PROGRAM AxisReset
VAR
END_VAR

//左臂
axis_LeftArm_Left_Reset(
	Axis:= axis_LeftArm_Left, 
	Execute:= bAxis_LeftArm_Left_Reset, 
	Done=> , 
	Busy=> , 
	Error=> , 
	ErrorID=> );
	
axis_LeftArm_Right_Reset(
	Axis:= axis_LeftArm_Right, 
	Execute:= bAxis_LeftArm_Right_Reset, 
	Done=> , 
	Busy=> , 
	Error=> , 
	ErrorID=> );

axis_LeftArm_Lift_Reset(
	Axis:= axis_LeftArm_Lift, 
	Execute:= bAxis_LeftArm_Lift_Reset, 
	Done=> , 
	Busy=> , 
	Error=> , 
	ErrorID=> );

axis_LeftArm_Wrist_Reset(
	Axis:= axis_LeftArm_Wrist, 
	Execute:= bAxis_LeftArm_Wrist_Reset, 
	Done=> , 
	Busy=> , 
	Error=> , 
	ErrorID=> );
	

//右臂
axis_RightArm_Left_Reset(
	Axis:= axis_RightArm_Left, 
	Execute:= bAxis_RightArm_Left_Reset, 
	Done=> , 
	Busy=> , 
	Error=> , 
	ErrorID=> );
	
axis_RightArm_Right_Reset(
	Axis:= axis_RightArm_Right, 
	Execute:= bAxis_RightArm_Right_Reset, 
	Done=> , 
	Busy=> , 
	Error=> , 
	ErrorID=> );

axis_RightArm_Lift_Reset(
	Axis:= axis_RightArm_Lift, 
	Execute:= bAxis_RightArm_Lift_Reset, 
	Done=> , 
	Busy=> , 
	Error=> , 
	ErrorID=> );

axis_RightArm_Wrist_Reset(
	Axis:= axis_RightArm_Wrist, 
	Execute:= bAxis_RightArm_Wrist_Reset, 
	Done=> , 
	Busy=> , 
	Error=> , 
	ErrorID=> );

//大龙门
axis_BigGate_Left_Reset(
	Axis:= axis_BigGate_Left, 
	Execute:= bAxis_BigGate_Left_Reset, 
	Done=> , 
	Busy=> , 
	Error=> , 
	ErrorID=> );
	
axis_BigGate_Right_Reset(
	Axis:= axis_BigGate_Right, 
	Execute:= bAxis_BigGate_Right_Reset, 
	Done=> , 
	Busy=> , 
	Error=> , 
	ErrorID=> );
	

//小龙门
axis_SmallGate_Left_Reset(
	Axis:= axis_SmallGate_Left, 
	Execute:= bAxis_SmallGate_Left_Reset, 
	Done=> , 
	Busy=> , 
	Error=> , 
	ErrorID=> );
	
axis_SmallGate_Right_Reset(
	Axis:= axis_SmallGate_Right, 
	Execute:= bAxis_SmallGate_Right_Reset, 
	Done=> , 
	Busy=> , 
	Error=> , 
	ErrorID=> );

	
	
//后龙门
axis_BackGate_Left_Reset(
	Axis:= axis_BackGate_Left, 
	Execute:= bAxis_BackGate_Left_Reset, 
	Done=> , 
	Busy=> , 
	Error=> , 
	ErrorID=> );
	
axis_BackGate_Right_Reset(
	Axis:= axis_BackGate_Right, 
	Execute:= bAxis_BackGate_Right_Reset, 
	Done=> , 
	Busy=> , 
	Error=> , 
	ErrorID=> );

END_PROGRAM

(* stored: Version 1.1.0.1, ProductVersion 3.1.4024.14
   POU AxisReset: Id {f0a21cb2-6fdb-47c3-b950-62c7b25507e5}, SpecialFunc None *)
